PROGRAM Background
VAR
END_VAR

BackgroundEL();

END_PROGRAM

(* stored: Version 1.1.0.1, ProductVersion 3.1.4024.11
   POU Background: Id {a474ab24-92b2-4faa-ab36-f1eb12602ab9}, SpecialFunc None *)
